// Mitsubishi GX Works2 project: 20150731_virtual_final8_test   PLC: Q02/Q02H

PROGRAM MAIN
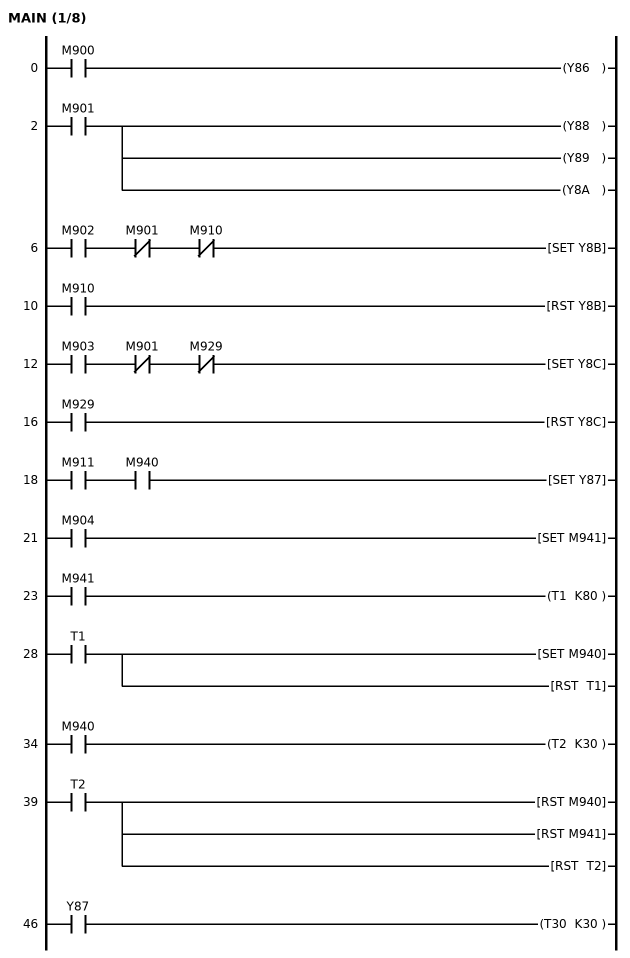
0     LD      M900
      OUT     Y86
2     LD      M901
      OUT     Y88
      OUT     Y89
      OUT     Y8A
6     LD      M902
      ANI     M901
      ANI     M910
      SET     Y8B
10    LD      M910
      RST     Y8B
12    LD      M903
      ANI     M901
      ANI     M929
      SET     Y8C
16    LD      M929
      RST     Y8C
18    LD      M911
      AND     M940
      SET     Y87
21    LD      M904
      SET     M941
23    LD      M941
      OUT     T1 K80
28    LD      T1
      SET     M940
      RST     T1
34    LD      M940
      OUT     T2 K30
39    LD      T2
      RST     M940
      RST     M941
      RST     T2
46    LD      Y87
      OUT     T30 K30
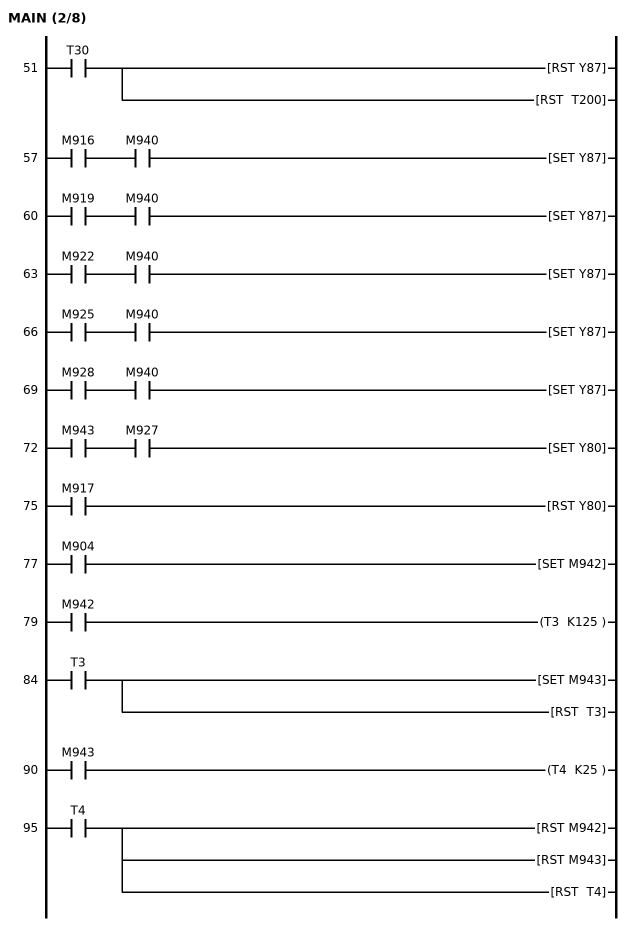
51    LD      T30
      RST     Y87
      RST     T200
57    LD      M916
      AND     M940
      SET     Y87
60    LD      M919
      AND     M940
      SET     Y87
63    LD      M922
      AND     M940
      SET     Y87
66    LD      M925
      AND     M940
      SET     Y87
69    LD      M928
      AND     M940
      SET     Y87
72    LD      M943
      AND     M927
      SET     Y80
75    LD      M917
      RST     Y80
77    LD      M904
      SET     M942
79    LD      M942
      OUT     T3 K125
84    LD      T3
      SET     M943
      RST     T3
90    LD      M943
      OUT     T4 K25
95    LD      T4
      RST     M942
      RST     M943
      RST     T4
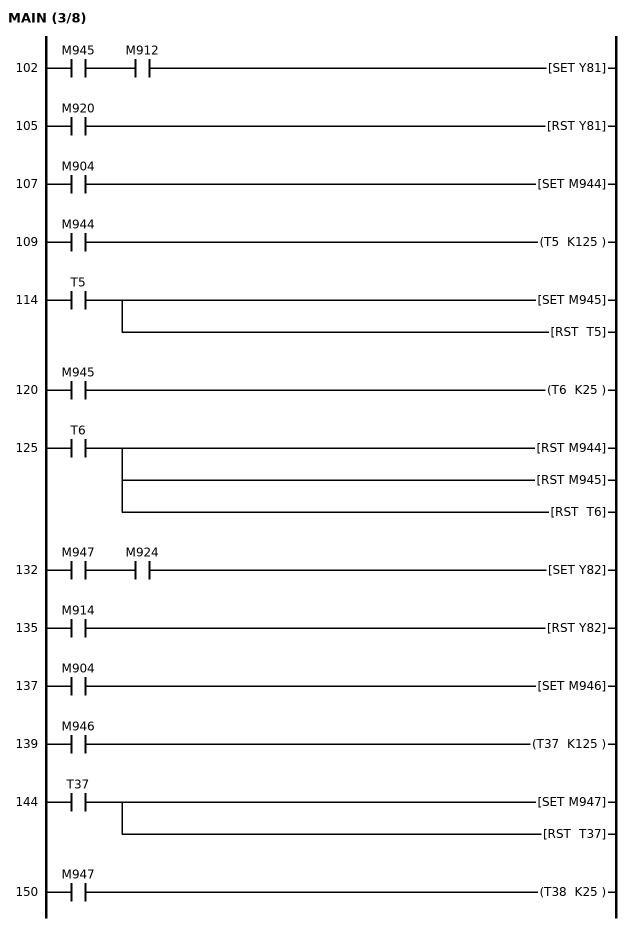
102   LD      M945
      AND     M912
      SET     Y81
105   LD      M920
      RST     Y81
107   LD      M904
      SET     M944
109   LD      M944
      OUT     T5 K125
114   LD      T5
      SET     M945
      RST     T5
120   LD      M945
      OUT     T6 K25
125   LD      T6
      RST     M944
      RST     M945
      RST     T6
132   LD      M947
      AND     M924
      SET     Y82
135   LD      M914
      RST     Y82
137   LD      M904
      SET     M946
139   LD      M946
      OUT     T37 K125
144   LD      T37
      SET     M947
      RST     T37
150   LD      M947
      OUT     T38 K25
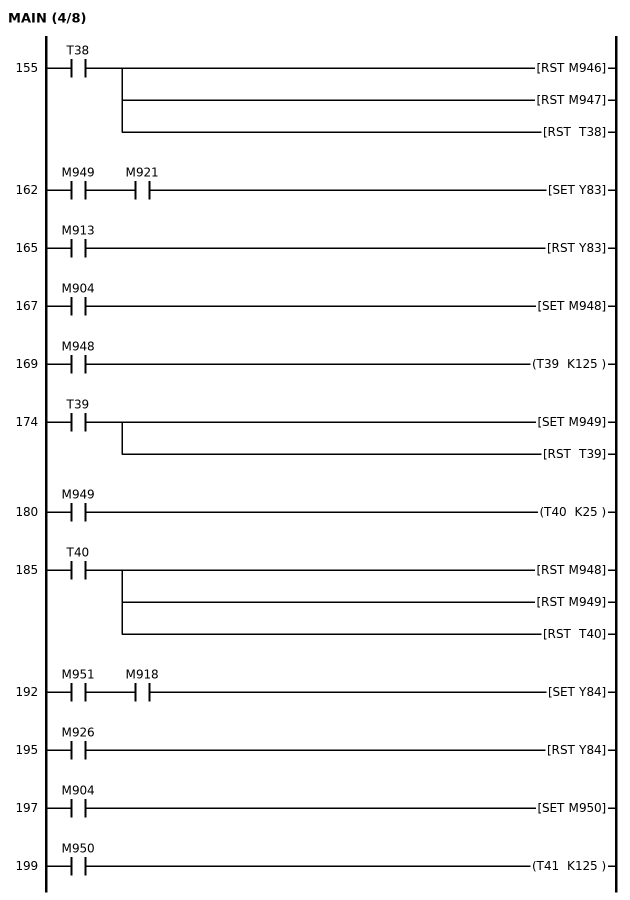
155   LD      T38
      RST     M946
      RST     M947
      RST     T38
162   LD      M949
      AND     M921
      SET     Y83
165   LD      M913
      RST     Y83
167   LD      M904
      SET     M948
169   LD      M948
      OUT     T39 K125
174   LD      T39
      SET     M949
      RST     T39
180   LD      M949
      OUT     T40 K25
185   LD      T40
      RST     M948
      RST     M949
      RST     T40
192   LD      M951
      AND     M918
      SET     Y84
195   LD      M926
      RST     Y84
197   LD      M904
      SET     M950
199   LD      M950
      OUT     T41 K125
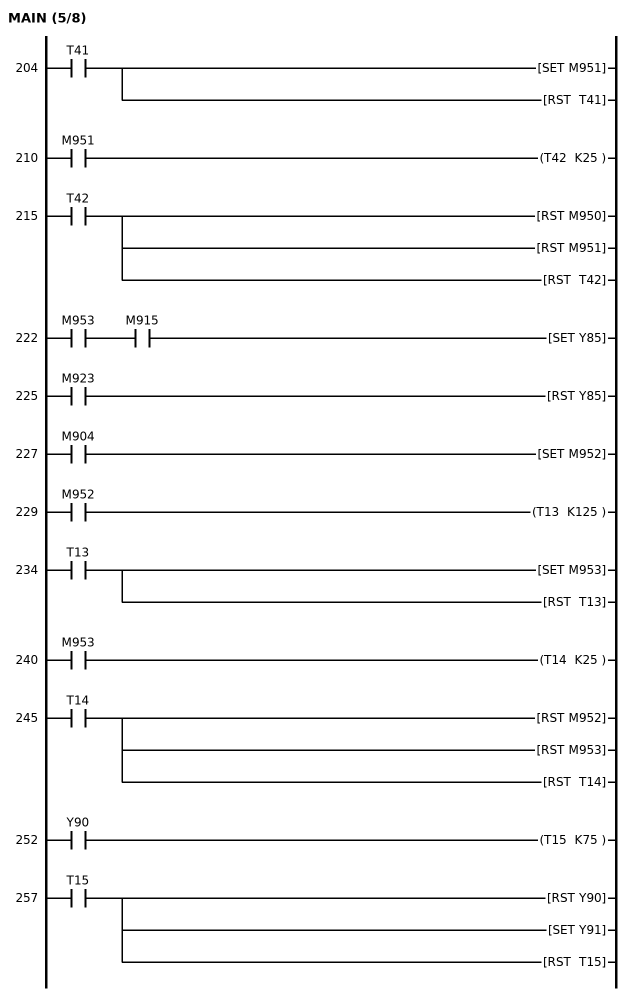
204   LD      T41
      SET     M951
      RST     T41
210   LD      M951
      OUT     T42 K25
215   LD      T42
      RST     M950
      RST     M951
      RST     T42
222   LD      M953
      AND     M915
      SET     Y85
225   LD      M923
      RST     Y85
227   LD      M904
      SET     M952
229   LD      M952
      OUT     T13 K125
234   LD      T13
      SET     M953
      RST     T13
240   LD      M953
      OUT     T14 K25
245   LD      T14
      RST     M952
      RST     M953
      RST     T14
252   LD      Y90
      OUT     T15 K75
257   LD      T15
      RST     Y90
      SET     Y91
      RST     T15
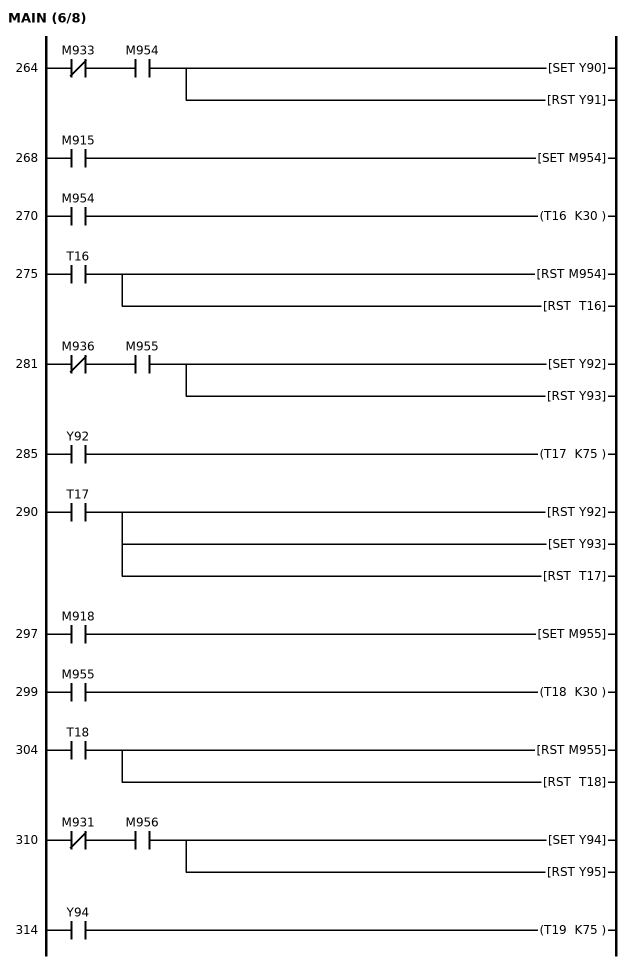
264   LDI     M933
      AND     M954
      SET     Y90
      RST     Y91
268   LD      M915
      SET     M954
270   LD      M954
      OUT     T16 K30
275   LD      T16
      RST     M954
      RST     T16
281   LDI     M936
      AND     M955
      SET     Y92
      RST     Y93
285   LD      Y92
      OUT     T17 K75
290   LD      T17
      RST     Y92
      SET     Y93
      RST     T17
297   LD      M918
      SET     M955
299   LD      M955
      OUT     T18 K30
304   LD      T18
      RST     M955
      RST     T18
310   LDI     M931
      AND     M956
      SET     Y94
      RST     Y95
314   LD      Y94
      OUT     T19 K75
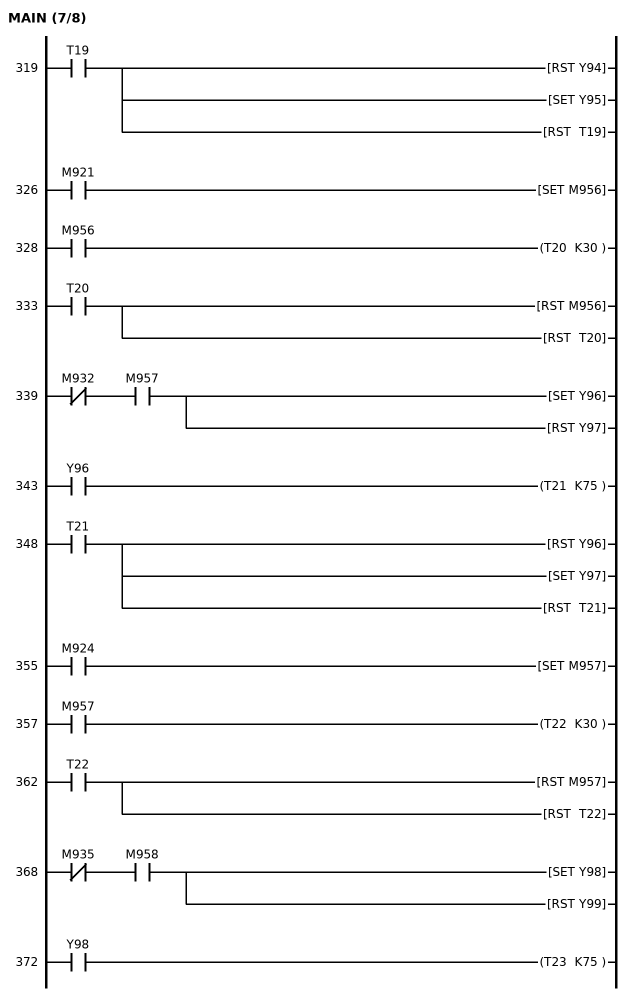
319   LD      T19
      RST     Y94
      SET     Y95
      RST     T19
326   LD      M921
      SET     M956
328   LD      M956
      OUT     T20 K30
333   LD      T20
      RST     M956
      RST     T20
339   LDI     M932
      AND     M957
      SET     Y96
      RST     Y97
343   LD      Y96
      OUT     T21 K75
348   LD      T21
      RST     Y96
      SET     Y97
      RST     T21
355   LD      M924
      SET     M957
357   LD      M957
      OUT     T22 K30
362   LD      T22
      RST     M957
      RST     T22
368   LDI     M935
      AND     M958
      SET     Y98
      RST     Y99
372   LD      Y98
      OUT     T23 K75
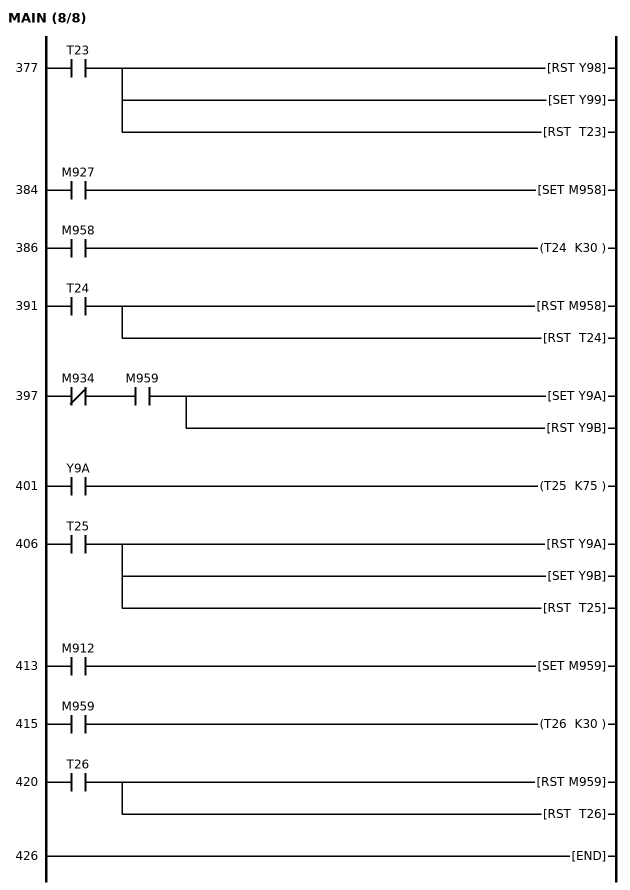
377   LD      T23
      RST     Y98
      SET     Y99
      RST     T23
384   LD      M927
      SET     M958
386   LD      M958
      OUT     T24 K30
391   LD      T24
      RST     M958
      RST     T24
397   LDI     M934
      AND     M959
      SET     Y9A
      RST     Y9B
401   LD      Y9A
      OUT     T25 K75
406   LD      T25
      RST     Y9A
      SET     Y9B
      RST     T25
413   LD      M912
      SET     M959
415   LD      M959
      OUT     T26 K30
420   LD      T26
      RST     M959
      RST     T26
426   END
END_PROGRAM
